INTERFACE I_AO_Voltage

PROPERTY errId : HAL_ErrorEnum
GET
END_GET
END_PROPERTY

PROPERTY rValue : real
GET
END_GET
SET
END_SET
END_PROPERTY

END_INTERFACE

(* stored: Version 1.1.0.1, ProductVersion 3.1.4024.6
   Itf I_AO_Voltage: Id {b485a4bc-c8f6-08a2-3418-5be1278f5119}
   Property errId: Id {2c4d432a-2787-00f0-1d0b-5d87567d5e59}
   Get Get: Id {b82f2e52-9aad-085b-03f1-cc63383c5bff}
   Property rValue: Id {c2ddfcb2-f0ae-0c89-227e-78092d387bf7}
   Get Get: Id {cb5d1f91-297c-0c37-0c0c-d7e8b8b6560c}
   Set Set: Id {b47cb871-8d64-0ce3-05b4-ebe974c63816} *)
